KUKA KRL program: RESET_VAR.src

&ACCESS RV
&PARAM EDITMASK = *
&PARAM TEMPLATE = C:\KRC\Roboter\Template\FunctionVorgabe
DEFFCT BOOL RESET_VAR( )

ENDFCT
